(* CoDeSys 2.3 export: APPLERRORNEW_TS.EXP *)

(* Data type in Diag/Error *)
TYPE ApplErrorNew_ts :
(* ApplError_ts *)
STRUCT
	Code_u16					: UINT;
	Description_as8		: STRING(32);
(*	Description_as8		: ARRAY [1..4] OF STRING(32);*)
END_STRUCT
END_TYPE
